Staubli VAL3: setPos.pgx

program setPos(num x_nAxisNum (dimensions=1), num x_nCurrentPos (dimensions=1))
begin
  //
  aioSet(aoPosCmd[x_nAxisNum],x_nCurrentPos)
end
